(* CODESYS project Untitled1.project

Project tree, tasks and I/O mapping:
  Device : CODESYS Control Win V3, 3S - Smart Software Solutions GmbH, order no. 305021, version 3.5.5.50
    application Application
      libraries: Standard, * (System)
      task MainTask (cyclic, interval t#100ms, priority 1) calls btn_release_prg
      task VISU_TASK (cyclic, interval 100 ms, priority 31) calls VisuElems.Visu_Prg
      task task_btn_push (event, event btn, priority 1) calls btn_push_prg
      task btn_period_task (event, event btn_peiod, priority 1) calls btn_period
      program task_one [ST]
      global variables GVL
      visualisation Visualization
      program task_two [ST]
      program btn_release_prg [ST]
      program btn_push_prg [ST]
      program btn_period [ST]
  text list GlobalTextList
*)

// Device/Application/GVL
VAR_GLOBAL
	co2_sensor: INT := 10;
	valve: BOOL := FALSE; // FALSE--> closed ; TRUE --> open
	valve_prop: INT := -24; // FALSE--> closed ; TRUE --> open
	btn: BOOL := FALSE; // FALSE--> closed ; TRUE --> open
	btn_peiod: BOOL := FALSE; // FALSE--> closed ; TRUE --> open
END_VAR

// Device/Application/btn_release_prg
PROGRAM btn_release_prg
VAR
	check_btn: F_TRIG; // detects HIGH --> LOW
END_VAR

VAR_OUTPUT
	Q: BOOL;
END_VAR

check_btn(CLK:=btn);

IF check_btn.Q = TRUE THEN
	valve:= FALSE;
END_IF

END_PROGRAM

// Device/Application/btn_push_prg
PROGRAM btn_push_prg
VAR
END_VAR

valve:=True;

END_PROGRAM

// Device/Application/btn_period
PROGRAM btn_period
VAR
	timer: TP;
	start_flag: BOOL;
	start: BOOL;
	BREAK: INT;
END_VAR

// 3 вида: таймер с задержкой включения, таймер с задержкой выключения, таймер периода
// T_ON, T_OFF, TP = time period
start_flag := TRUE;
valve := TRUE;
timer(in:=start_flag, pt:=T#5S);

WHILE TRUE DO
	timer(in:=start_flag, pt:=T#5S);
	IF timer.Q = FALSE THEN
		start_flag := FALSE;
		valve:=FALSE;
		timer(in:=start_flag, pt:=T#5S);
		EXIT;
	END_IF
END_WHILE

END_PROGRAM

// Device/Application/task_one
PROGRAM task_one
VAR
	MAX_LIMIT: INT := 25;
	MIN_LIMIT: INT := 15;
END_VAR

IF co2_sensor > MAX_LIMIT THEN
	valve:= FALSE;
ELSIF co2_sensor  < MIN_LIMIT THEN
	valve:= TRUE;
END_IF

END_PROGRAM

// Device/Application/task_two
PROGRAM task_two
VAR
	MIN_CO2: INT := 0;
	MAX_CO2: INT := 30;
	MIN_VALVE: INT:= -24;
	MAX_VALVE: INT:= 24;
END_VAR

// arduino map --> function
// valve_prop := (x - in_min) * (out_max - out_min) / (in_max - in_min) + out_min;
IF co2_sensor > MAX_CO2 THEN
	valve_prop:=MAX_VALVE;
ELSE 
	valve_prop := -(  (co2_sensor - MIN_CO2) * (MAX_VALVE - MIN_VALVE) / (MAX_CO2 - MIN_CO2) + MIN_VALVE );
END_IF

END_PROGRAM

// Device/Application/Visualization
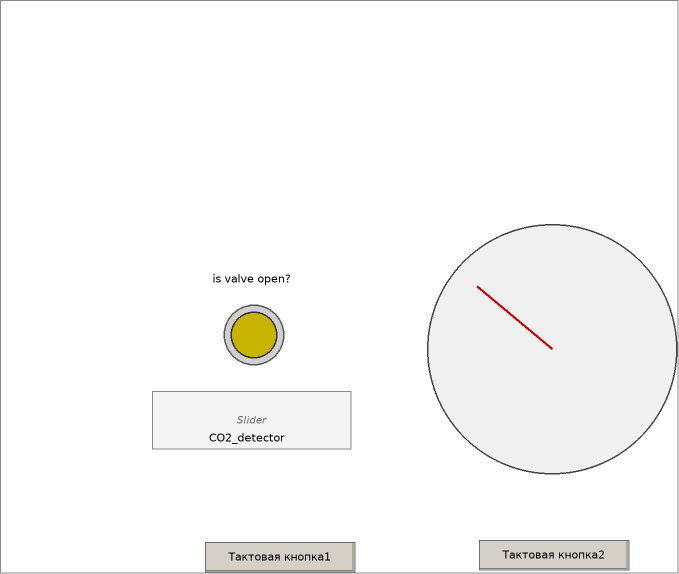
VISUALIZATION Visualization  // 679x574
    Slider (152,391 199x58), variable: co2_sensor, scale 0..30
    Label (172,423 150x30), "CO2_detector"
    Lamp1 (219,300 70x70), variable: valve, style: Lamp-Lamp1-Yellow
    Label (177,264 150x30), "is valve open?"
    Meter360 (427,224 250x250), value: valve_prop, style: Meter-Meter360-Gray, scale format: %.1f, scale -24..24
    Button (205,542 150x30), "Тактовая кнопка1"
        tap btn
    Button (479,540 150x30), "Тактовая кнопка2"
        tap btn_peiod
END_VISUALIZATION
